// TIA Portal V16 export
// export: Created 2021-11-12T13:32:48.1042849Z, ExportSetting WithDefaults, DisplayName Totally Integrated Automation Portal, DisplayVersion V16 Update 3, DisplayName TIA Portal Version Control Interface, DisplayVersion V16 Update 2, DisplayName TIA Portal Openness, DisplayVersion V16 Update 3, DisplayName SINAMICS Startdrive Advanced, DisplayVersion V16 Update 5, DisplayName SINAMICS Startdrive G130, G150, S120, S150, SINAMICS MV, S210, DisplayVersion V16 Update 5, DisplayName SINAMICS Startdrive G110M, G120, G120C, G120D, G120P, G115D, DisplayVersion V16 Update 5, DisplayName STEP 7 Professional, DisplayVersion V16 Update 3, DisplayName STEP 7 Safety, DisplayVersion V16, DisplayName WinCC UA Professional, DisplayVersion V16 Update 3
DATA_BLOCK "IDB_Station330"   // DB196
VERSION : 0.1
// stored: AutoNumber true, DBAccessibleFromOPCUA true, InstanceOfName Station330, InstanceOfType FB
"Station330"
   // VAR
   //    SF_CL01_Alarm { S7_SetPoint := 'True'} : "STD_DI_Mon";
   //    SF_CL01_Warning { S7_SetPoint := 'True'} : "STD_DI_Mon";
   //    SF_GL01_MA1 : "STD_Drive1";
   //    SF_GL02_MA1 { S7_SetPoint := 'True'} : "STD_Drive1";
   //    SF_GL03_MA1 { S7_SetPoint := 'True'} : "STD_Drive1";
   //    SF_UC21_TA1 { S7_SetPoint := 'True'} : "STD_Siemens_G120_CU240E_2_PN";
   //    SF_UC21_TA2 { S7_SetPoint := 'True'} : "STD_Siemens_G120_CU240E_2_PN";
   //    SF_UC21_TA3 { S7_SetPoint := 'True'} : "STD_Siemens_G120_CU240E_2_PN";
   //    SF_TON_1 { S7_SetPoint := 'True'} : TON_TIME;
   //    SB1_PowerOk { S7_SetPoint := 'True'} : Bool;
   //    SF_BoxPartCounter { S7_SetPoint := 'True'} : "STD_PartCounter";
   //    SB1BoxExchangeReq { S7_SetPoint := 'True'} : Bool;
   //    ST_TOF320_GL01_1Tact { S7_SetPoint := 'True'} : TOF_TIME;
   //    ST_TOF320_GL01_2Tact { S7_SetPoint := 'True'} : TOF_TIME;
   //    ST_TOF330_GL01Tact { S7_SetPoint := 'True'} : TOF_TIME;
   //    ST_TOF330_GL02Tact { S7_SetPoint := 'True'} : TOF_TIME;
   // END_VAR
BEGIN
END_DATA_BLOCK
